TEXTLIST MachineType
  0 = 'None'
  1 = '367' | Chinese: '367' | English: '367' | Vietnamese: '367'
  2 = '201' | Chinese: '201' | English: '201' | Vietnamese: '201'
  3 = '373' | Chinese: '373' | English: '373' | Vietnamese: '373'
  4 = '69' | Chinese: '69' | English: '69' | Vietnamese: '69'
  5 = '311' | Chinese: '311' | English: '311' | Vietnamese: '311'
   = ''
END_TEXTLIST

(* stored: Version 1.1.0.1, ProductVersion 3.1.4024.3
   TextList MachineType: Id {47a7ad8a-9585-4eca-9473-fcd62ad043b5} *)
